// TIA Portal V20 export
TYPE "typeCmControlNodeBrakeTest"
// stored: Namespace Unit1.Em7
   STRUCT
      ngKicker { ExternalWritable := 'False'} : "LER_typeBrakeTestEmControlNodes";
      passKicker { ExternalWritable := 'False'} : "LER_typeBrakeTestEmControlNodes";
   END_STRUCT;
END_TYPE
